// TIA Portal project "PID_Tank_V17" (V17)

(* hardware
DEVICE "S7-1200 station_1"  S7-1200 Station
   slot 0: "Rack_0"  S7-1200 Rack  Rack  V1.0
   slot 1: "PLC_1"  CPU 1215C DC/DC/DC  6ES7 215-1AG40-0XB0  V4.4
DEVICE "HMI_1"  KTP700 Basic PN
   slot 0: "HMI_1"  KTP700 Basic PN  6AV2 123-2GB03-0AX0  16.0.0.0
   slot 1: "HMI_RT_1"  KTP700 Basic PN  6AV2 123-2GB03-0AX0  16.0.0.0
   slot 5: "HMI_1.IE_CP_1"  PROFINET Interface  16.0.0.0
      slot 1: "PROFINET Interface_1"  PROFINET Interface
         slot 1: "Port_1"  Port
*)

// ===== PLC "PLC_1"  CPU 1215C DC/DC/DC =====

VAR_GLOBAL   // PLC tag table "Default tag table"
   "IW_TankLevel_Sensor" AT %ID30 : Real;
   "IW_Flow_Sensor" AT %ID34 : Real;
   "Q_Hooter" AT %Q0.0 : Bool;
   "QW_DrainValve_Signal" AT %QD34 : Real;
   "QW_FillingValve_Signal" AT %QD30 : Real;
END_VAR

DATA_BLOCK "FB_PID_DB"   // DB5
{ S7_Optimized_Access := 'TRUE' }
VERSION : 0.1
// stored: InstanceOfName FB_PID
"FB_PID"
BEGIN
END_DATA_BLOCK

// folder: Global DB

DATA_BLOCK "DB_System"   // DB2
{ S7_Optimized_Access := 'TRUE' }
VERSION : 0.1
   VAR
      "ActualValue_%" : Real;
      "ProcessVAlue_PV_%" : Real;
   END_VAR
BEGIN
END_DATA_BLOCK

DATA_BLOCK "DB_Alarm"   // DB3
{ S7_Optimized_Access := 'TRUE' }
VERSION : 0.1
BEGIN
END_DATA_BLOCK

DATA_BLOCK "DB_HMI_Interface"   // DB4
{ S7_Optimized_Access := 'TRUE' }
VERSION : 0.1
   VAR
      From_HMI_To_PLC : Struct
         "SetValue_SP_%" : Real;
         ki : Real;
         kp : Real;
         kd : Real;
         Auto : Bool;
         DrainValve_SetPoint : Real;
         AlarmBit : Bool;
      END_STRUCT;
      From_PLC_To_HMI : Struct
         ActualValue : Real;
         SetValue_SP_InRange : Real;
         "ActualValue_%" : Real;
         "Error_%" : Real;
         Error_InRange : Real;
         Filling_Pipe_Animation_SetPoint : Int;
         P_Term : Real;
         I_Term : Real;
         D_Term : Real;
         FillingValve_SetPoint : Real;
      END_STRUCT;
      Alarm : Word;
   END_VAR
BEGIN
END_DATA_BLOCK

// folder: IO_mapping

DATA_BLOCK "DB_IO_Mapping"   // DB1
{ S7_Optimized_Access := 'TRUE' }
VERSION : 0.1
   VAR
      Input : Struct
         IW_TankLevel_Sensor : Real;
         IW_Flow_Sensor : Real;
      END_STRUCT;
      Output : Struct
         Q_Hooter : Bool;
         QW_DrainValve_Signal : Real;
         QW_FillingValve_Signal : Real;
      END_STRUCT;
   END_VAR
BEGIN
END_DATA_BLOCK

// folder: (top level)

ORGANIZATION_BLOCK "Main"   // OB1, LAD, ProgramCycle
TITLE = "Main Program Sweep (Cycle)"
{ S7_Optimized_Access := 'TRUE' }
VERSION : 0.1
   VAR_INPUT
      Initial_Call : Bool;   // Initial call of this OB
      Remanence : Bool;   // =True, if remanent data are available
   END_VAR
BEGIN

REGION Network 1: Factory IO Connection
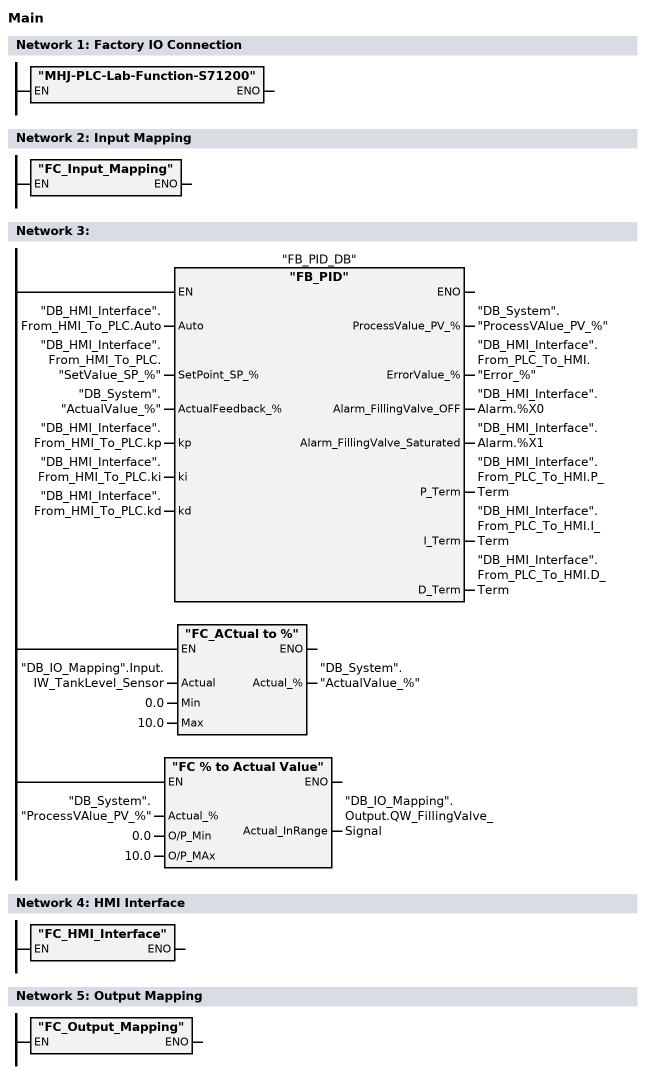
   RUNG wire#powerrail
      "MHJ-PLC-Lab-Function-S71200"()
   END_RUNG
   // the same network as SCL:
   "MHJ-PLC-Lab-Function-S71200"();
END_REGION

REGION Network 2: Input Mapping
   RUNG wire#powerrail
      "FC_Input_Mapping"()
   END_RUNG
   // the same network as SCL:
   "FC_Input_Mapping"();
END_REGION

REGION Network 3
   RUNG wire#powerrail
      "FB_PID_DB"(Auto := "DB_HMI_Interface".From_HMI_To_PLC.Auto, "SetPoint_SP_%" := "DB_HMI_Interface".From_HMI_To_PLC."SetValue_SP_%", "ActualFeedback_%" := "DB_System"."ActualValue_%", kp := "DB_HMI_Interface".From_HMI_To_PLC.kp, ki := "DB_HMI_Interface".From_HMI_To_PLC.ki, kd := "DB_HMI_Interface".From_HMI_To_PLC.kd, "ProcessValue_PV_%" => "DB_System"."ProcessVAlue_PV_%", "ErrorValue_%" => "DB_HMI_Interface".From_PLC_To_HMI."Error_%", Alarm_FillingValve_OFF => "DB_HMI_Interface".Alarm.%X0, Alarm_FillingValve_Saturated => "DB_HMI_Interface".Alarm.%X1, P_Term => "DB_HMI_Interface".From_PLC_To_HMI.P_Term, I_Term => "DB_HMI_Interface".From_PLC_To_HMI.I_Term, D_Term => "DB_HMI_Interface".From_PLC_To_HMI.D_Term)
   END_RUNG
   RUNG wire#powerrail
      "FC_ACtual to %"(Actual := "DB_IO_Mapping".Input.IW_TankLevel_Sensor, Min := 0.0, Max := 10.0, "Actual_%" => "DB_System"."ActualValue_%")
   END_RUNG
   RUNG wire#powerrail
      "FC % to Actual Value"("Actual_%" := "DB_System"."ProcessVAlue_PV_%", "O/P_Min" := 0.0, "O/P_MAx" := 10.0, Actual_InRange => "DB_IO_Mapping".Output.QW_FillingValve_Signal)
   END_RUNG
   // the same network as SCL:
   "FB_PID_DB"(Auto := "DB_HMI_Interface".From_HMI_To_PLC.Auto,   // "FB_PID"
               "SetPoint_SP_%" := "DB_HMI_Interface".From_HMI_To_PLC."SetValue_SP_%",
               "ActualFeedback_%" := "DB_System"."ActualValue_%",
               kp := "DB_HMI_Interface".From_HMI_To_PLC.kp,
               ki := "DB_HMI_Interface".From_HMI_To_PLC.ki,
               kd := "DB_HMI_Interface".From_HMI_To_PLC.kd,
               "ProcessValue_PV_%" => "DB_System"."ProcessVAlue_PV_%",
               "ErrorValue_%" => "DB_HMI_Interface".From_PLC_To_HMI."Error_%",
               Alarm_FillingValve_OFF => "DB_HMI_Interface".Alarm.%X0,
               Alarm_FillingValve_Saturated => "DB_HMI_Interface".Alarm.%X1,
               P_Term => "DB_HMI_Interface".From_PLC_To_HMI.P_Term,
               I_Term => "DB_HMI_Interface".From_PLC_To_HMI.I_Term,
               D_Term => "DB_HMI_Interface".From_PLC_To_HMI.D_Term);
   "FC_ACtual to %"(Actual := "DB_IO_Mapping".Input.IW_TankLevel_Sensor,
                    Min := 0.0,
                    Max := 10.0,
                    "Actual_%" => "DB_System"."ActualValue_%");
   "FC % to Actual Value"("Actual_%" := "DB_System"."ProcessVAlue_PV_%",
                          "O/P_Min" := 0.0,
                          "O/P_MAx" := 10.0,
                          Actual_InRange => "DB_IO_Mapping".Output.QW_FillingValve_Signal);
END_REGION

REGION Network 4: HMI Interface
   RUNG wire#powerrail
      "FC_HMI_Interface"()
   END_RUNG
   // the same network as SCL:
   "FC_HMI_Interface"();
END_REGION

REGION Network 5: Output Mapping
   RUNG wire#powerrail
      "FC_Output_Mapping"()
   END_RUNG
   // the same network as SCL:
   "FC_Output_Mapping"();
END_REGION
END_ORGANIZATION_BLOCK

// folder: FB_Library

FUNCTION_BLOCK "FB_PID"   // FB1, SCL
{ S7_Optimized_Access := 'TRUE' }
VERSION : 0.1
   VAR_INPUT
      Auto : Bool;
      "SetPoint_SP_%" : Real;
      "ActualFeedback_%" : Real;
      kp : Real;
      ki : Real;
      kd : Real;
   END_VAR
   VAR_OUTPUT
      "ProcessValue_PV_%" : Real;
      "ErrorValue_%" : Real;
      Alarm_FillingValve_OFF : Bool;
      Alarm_FillingValve_Saturated : Bool;
      P_Term : Real;
      I_Term : Real;
      D_Term : Real;
   END_VAR
   VAR
      Prev_Error : Real;
      IntegralError : Real;
      IntegralReset : Bool;
      FiilingValve_OFF_TONStart_Condition : Bool;
      FillingValve_Saturated_TONStart_Condition : Bool;
      IEC_Timer_0_Instance_FillingValve_OFF : TON_TIME;
      IEC_Timer_0_Instance_FillingValve_Saturated : TON_TIME;
   END_VAR
   VAR_TEMP
      p_Term_Temp : Real;
      i_Term_Temp : Real;
      d_Term_Temp : Real;
      Current_Error_Temp : Real;
      processed_Value_Temp : Real;
   END_VAR
BEGIN


   IF #Auto THEN

       #Current_Error_Temp :=  #"SetPoint_SP_%" - #"ActualFeedback_%" ;

       //P-Term Calculation
       #p_Term_Temp:= #Current_Error_Temp * #kp;

       //I-Term Calculation
       #i_Term_Temp := (#IntegralError + #Current_Error_Temp) * #ki;

       //D-Term Calculation
       #d_Term_Temp := ( #Current_Error_Temp - #Prev_Error) * #kd;

       //Process Value
       #processed_Value_Temp  := #p_Term_Temp + #i_Term_Temp + #d_Term_Temp;

       //Make Range 0-100
       IF #processed_Value_Temp > 100 THEN
           #processed_Value_Temp := 100;
       ELSIF #processed_Value_Temp < 0 THEN
           #processed_Value_Temp := 0;
       END_IF;


       //Alarm Detection

       //Filling Valve OFF
       IF (#"ActualFeedback_%" < #"SetPoint_SP_%") & (#Current_Error_Temp >= #Prev_Error) THEN
           #FiilingValve_OFF_TONStart_Condition := TRUE;
       ELSE
           #FiilingValve_OFF_TONStart_Condition := FALSE;
       END_IF;

       //Make timer On or OFF
       IF #FiilingValve_OFF_TONStart_Condition THEN
           #IEC_Timer_0_Instance_FillingValve_OFF(IN:=TRUE,
                         PT:=T#30s);
       ELSE
           #IEC_Timer_0_Instance_FillingValve_OFF(IN := FALSE,
                                 PT := T#30s);
       END_IF;
       //IF timer On than Set Alarm
       IF #IEC_Timer_0_Instance_FillingValve_OFF.Q THEN
           #Alarm_FillingValve_OFF := TRUE;
       ELSE
           #Alarm_FillingValve_OFF := FALSE;
       END_IF;

       //Filling Valve Saturated Alarm
       IF (#"ActualFeedback_%" > #"SetPoint_SP_%") & (#Current_Error_Temp <= #Prev_Error) THEN
           #FillingValve_Saturated_TONStart_Condition := TRUE;
       ELSE
           #FillingValve_Saturated_TONStart_Condition := FALSE;
       END_IF;

       IF #FillingValve_Saturated_TONStart_Condition THEN
           #IEC_Timer_0_Instance_FillingValve_Saturated(IN := TRUE,
                                                        PT := T#30s);
       ELSE
           #IEC_Timer_0_Instance_FillingValve_Saturated(IN := FALSE,
                                                        PT := T#30s);
       END_IF;

       IF #IEC_Timer_0_Instance_FillingValve_Saturated.Q THEN
           #Alarm_FillingValve_Saturated := TRUE;
       ELSE
           #Alarm_FillingValve_Saturated := FALSE;
       END_IF;



       //------------------------
       //Write to O/P
       #"ProcessValue_PV_%" := #processed_Value_Temp;
       #"ErrorValue_%" := #Current_Error_Temp;
       #P_Term := #p_Term_Temp;
       #I_Term := #i_Term_Temp;
       #D_Term := #d_Term_Temp;

       //Write State data
       #Prev_Error := #Current_Error_Temp;
       #IntegralError := #IntegralError + #Current_Error_Temp;


   ELSE
       #IntegralError := 0;
       #Prev_Error := 0;
       #IntegralReset := 0;
       #FiilingValve_OFF_TONStart_Condition := FALSE;
       #FillingValve_Saturated_TONStart_Condition := FALSE;
       #"ProcessValue_PV_%" := 0;
       #P_Term := 0;
       #I_Term := 0;
       #D_Term := 0;
       #Alarm_FillingValve_OFF := FALSE;
       #Alarm_FillingValve_Saturated := FALSE;
   END_IF;
END_FUNCTION_BLOCK

// folder: FC_Library

FUNCTION "FC_HMI_Interface" : Void   // FC3, SCL
{ S7_Optimized_Access := 'TRUE' }
VERSION : 0.1
   VAR_TEMP
      Norm_Data : Real;
   END_VAR
BEGIN

   #Norm_Data := NORM_X(MIN := 0.0, VALUE := "DB_IO_Mapping".Input.IW_TankLevel_Sensor, MAX := 10.0);

   "DB_HMI_Interface".From_PLC_To_HMI.ActualValue := SCALE_X(MIN := 0.0, VALUE := #Norm_Data, MAX := 300.0);
   "DB_HMI_Interface".From_PLC_To_HMI.Filling_Pipe_Animation_SetPoint := REAL_TO_INT("DB_HMI_Interface".From_PLC_To_HMI.ActualValue);
   "DB_HMI_Interface".From_PLC_To_HMI."ActualValue_%" := SCALE_X(MIN := 0.0, VALUE := #Norm_Data, MAX := 100.0);

   IF "DB_HMI_Interface".From_HMI_To_PLC.Auto THEN
       "DB_IO_Mapping".Output.QW_DrainValve_Signal := "DB_HMI_Interface".From_HMI_To_PLC.DrainValve_SetPoint;
   ELSE
       "DB_IO_Mapping".Output.QW_DrainValve_Signal := 0.0;
   END_IF;
   "DB_HMI_Interface".From_PLC_To_HMI.SetValue_SP_InRange := SCALE_X(MIN := 0.0, VALUE := "DB_HMI_Interface".From_HMI_To_PLC."SetValue_SP_%", MAX := 3.0);
   "DB_HMI_Interface".From_PLC_To_HMI."ActualValue_%" := "DB_System"."ActualValue_%";
   "DB_HMI_Interface".From_PLC_To_HMI.Error_InRange := SCALE_X(MIN := 0.0, VALUE := "DB_HMI_Interface".From_PLC_To_HMI."Error_%" , MAX := 3.0);

   "DB_HMI_Interface".From_PLC_To_HMI.FillingValve_SetPoint := "DB_IO_Mapping".Output.QW_FillingValve_Signal;

   "DB_IO_Mapping".Output.Q_Hooter := "DB_HMI_Interface".From_HMI_To_PLC.AlarmBit;
END_FUNCTION

FUNCTION "FC_ACtual to %" : Void   // FC4, SCL
{ S7_Optimized_Access := 'TRUE' }
VERSION : 0.1
   VAR_INPUT
      Actual : Real;
      Min : Real;
      Max : Real;
   END_VAR
   VAR_OUTPUT
      "Actual_%" : Real;
   END_VAR
   VAR_TEMP
      Norm_Value : Real;
   END_VAR
BEGIN
   #Norm_Value:=NORM_X(MIN:=#Min, VALUE:=#Actual, MAX:=#Max);
   #"Actual_%" := SCALE_X(MIN := 0.0, VALUE := #Norm_Value, MAX := 100.0);
END_FUNCTION

FUNCTION "FC % to Actual Value" : Void   // FC5, SCL
{ S7_Optimized_Access := 'TRUE' }
VERSION : 0.1
   VAR_INPUT
      "Actual_%" : Real;
      "O/P_Min" : Real;
      "O/P_MAx" : Real;
   END_VAR
   VAR_OUTPUT
      Actual_InRange : Real;
   END_VAR
   VAR_TEMP
      Norm_Value : Real;
   END_VAR
BEGIN
   #Norm_Value := NORM_X(MIN := 0.0, VALUE := #"Actual_%", MAX := 100.0);
   #Actual_InRange := SCALE_X(MIN := #"O/P_Min", VALUE := #Norm_Value, MAX := #"O/P_MAx");
END_FUNCTION

FUNCTION "MHJ-PLC-Lab-Function-S71200" : Void   // FC9000, SCL
{ S7_Optimized_Access := 'TRUE' }
VERSION : 0.1
   VAR_TEMP
      rdTimeReturn : Int;
      outputTime : DTL;
      SyncVal : Byte;
      forVal : Int;
      forVal_2 : Int;
      Value : Byte;
   END_VAR
   VAR CONSTANT
      CompVal : Byte := 16#34;
      Value_01 : Byte := 16#11;
      Value_01_DW : DWord := 16#A165_D992;
      Value_02_DW : DWord := 16#58BE_4401;
   END_VAR
BEGIN

   #Value:=PEEK(area := 16#82,
        dbNumber := 0,
        byteOffset := 511);
   #Value := #Value + 1;

   POKE(area := 16#82,
        dbNumber := 0,
        byteOffset := 511,
        value := #Value);

   POKE(area:=16#81,
        dbNumber:=0,
        byteOffset:=1016,
        value:=#Value_01_DW);
   POKE(area := 16#81,
        dbNumber := 0,
        byteOffset := 1020,
        value := #Value_02_DW);

   POKE(area := 16#81,
        dbNumber := 0,
        byteOffset := 511,
        value := B#16#00);

   FOR #forVal := 0 TO 500 DO
       FOR #forVal_2:=0 TO 10 DO
           #rdTimeReturn:=RD_SYS_T(#outputTime);
           #rdTimeReturn := WR_SYS_T(#outputTime);
           #rdTimeReturn := RD_SYS_T(#outputTime);
           #rdTimeReturn := WR_SYS_T(#outputTime);
       END_FOR;
       #SyncVal:= PEEK(area := 16#81,
                      dbNumber := 0,
                      byteOffset := 511);
       IF #SyncVal = #CompVal THEN
          GOTO M_1;
       END_IF;
   END_FOR;
   RETURN;

   M_1:
   POKE(area := 16#81,
        dbNumber := 0,
        byteOffset := 511,
        value := B#16#0);
END_FUNCTION

// folder: IO_mapping

FUNCTION "FC_Input_Mapping" : Void   // FC1, SCL
{ S7_Optimized_Access := 'TRUE' }
VERSION : 0.1
   VAR_TEMP
      ScaledData : Real;
   END_VAR
BEGIN

   "DB_IO_Mapping".Input.IW_TankLevel_Sensor := "IW_TankLevel_Sensor";
   "DB_IO_Mapping".Input.IW_Flow_Sensor := "IW_Flow_Sensor";
END_FUNCTION

FUNCTION "FC_Output_Mapping" : Void   // FC2, SCL
{ S7_Optimized_Access := 'TRUE' }
VERSION : 0.1
BEGIN

   "Q_Hooter" := "DB_IO_Mapping".Output.Q_Hooter;
   "QW_DrainValve_Signal" := "DB_IO_Mapping".Output.QW_DrainValve_Signal;
   "QW_FillingValve_Signal" := "DB_IO_Mapping".Output.QW_FillingValve_Signal;
END_FUNCTION

(* ===== HMI "HMI_RT_1" =====
system functions are stored by id; their names below are inferred from use
connection "HMI_Connection_1": ETHERNET, SMART_S7_1200_OMS

HMI tags "Default tag table"
   "Tag_ScreenNumber" : UInt, internal
   "DB_HMI_Interface_From_HMI_To_PLC_SetValue_SP_%" : Real = PLC DB_HMI_Interface.From_HMI_To_PLC.SetValue_SP_%, 1 s
   "DB_HMI_Interface_From_PLC_To_HMI_ActualValue_%" : Real = PLC DB_HMI_Interface.From_PLC_To_HMI.ActualValue_%, 1 s
   "DB_HMI_Interface_From_PLC_To_HMI_ActualValue_PV" : Real = PLC DB_HMI_Interface.From_PLC_To_HMI.ActualValue, 1 s
   "DB_HMI_Interface_From_PLC_To_HMI_Error_%" : Real = PLC DB_HMI_Interface.From_PLC_To_HMI.Error_%, 1 s
   "DB_HMI_Interface_From_PLC_To_HMI_Error_InRange" : Real = PLC DB_HMI_Interface.From_PLC_To_HMI.Error_InRange, 1 s
   "DB_HMI_Interface_From_HMI_To_PLC_ki" : Real = PLC DB_HMI_Interface.From_HMI_To_PLC.ki, 1 s
   "DB_HMI_Interface_From_HMI_To_PLC_kp" : Real = PLC DB_HMI_Interface.From_HMI_To_PLC.kp, 1 s
   "DB_HMI_Interface_From_HMI_To_PLC_kd" : Real = PLC DB_HMI_Interface.From_HMI_To_PLC.kd, 1 s
   "DB_HMI_Interface_From_HMI_To_PLC_DrainValve_SetPoint" : Real = PLC DB_HMI_Interface.From_HMI_To_PLC.DrainValve_SetPoint, 1 s
   "DB_HMI_Interface_From_HMI_To_PLC_Auto" : Bool = PLC DB_HMI_Interface.From_HMI_To_PLC.Auto, 1 s
   "DB_HMI_Interface_From_PLC_To_HMI_SetValue_SP_InRange" : Real = PLC DB_HMI_Interface.From_PLC_To_HMI.SetValue_SP_InRange, 100 ms
   "DB_HMI_Interface_From_PLC_To_HMI_Filling_Valve_SetPoint" : Int = PLC DB_HMI_Interface.From_PLC_To_HMI.Filling_Pipe_Animation_SetPoint, 1 s
   "DB_HMI_Interface_From_PLC_To_HMI_FillingValve_SetPoint" : Real = PLC DB_HMI_Interface.From_PLC_To_HMI.FillingValve_SetPoint, 1 s
   "DB_HMI_Interface_From_PLC_To_HMI_P_Term" : Real = PLC DB_HMI_Interface.From_PLC_To_HMI.P_Term, 1 s
   "DB_HMI_Interface_From_PLC_To_HMI_I_Term" : Real = PLC DB_HMI_Interface.From_PLC_To_HMI.I_Term, 1 s
   "DB_HMI_Interface_From_PLC_To_HMI_D_Term" : Real = PLC DB_HMI_Interface.From_PLC_To_HMI.D_Term, 1 s
   "DB_HMI_Interface_Alarm" : Word = PLC DB_HMI_Interface.Alarm, 1 s
   "DB_HMI_Interface_From_HMI_To_PLC_AlarmBit" : Bool = PLC DB_HMI_Interface.From_HMI_To_PLC.AlarmBit, 1 s

discrete alarms
   1: 'Filling Valve Failure Detected- Valave OFF', class Errors, trigger "DB_HMI_Interface_Alarm" bit 0
      on Coming: SetBit("DB_HMI_Interface_From_HMI_To_PLC_AlarmBit")
      on Going: ResetBit("DB_HMI_Interface_From_HMI_To_PLC_AlarmBit")
      on Acknowledge: ResetBit("DB_HMI_Interface_From_HMI_To_PLC_AlarmBit")
   2: 'Filling Valve Failure Detected- Valave Saturated', class Errors, trigger "DB_HMI_Interface_Alarm" bit 1
      on Coming: SetBit("DB_HMI_Interface_From_HMI_To_PLC_AlarmBit")
      on Going: ResetBit("DB_HMI_Interface_From_HMI_To_PLC_AlarmBit")
      on Acknowledge: ResetBit("DB_HMI_Interface_From_HMI_To_PLC_AlarmBit")

analog alarms
   1: 'Level High Detected', class Warnings, trigger "DB_HMI_Interface_From_PLC_To_HMI_ActualValue_%"
   2: 'Level Critical High Detected', class Errors, trigger "DB_HMI_Interface_From_PLC_To_HMI_ActualValue_%"
      on Coming: SetBit("DB_HMI_Interface_From_HMI_To_PLC_AlarmBit")
      on Going: ResetBit("DB_HMI_Interface_From_HMI_To_PLC_AlarmBit")
      on Acknowledge: ResetBit("DB_HMI_Interface_From_HMI_To_PLC_AlarmBit")
   3: 'Level Low Detected', class Warnings, trigger "DB_HMI_Interface_From_PLC_To_HMI_ActualValue_%"
   4: 'Level Critical Low Detected', class Errors, trigger "DB_HMI_Interface_From_PLC_To_HMI_ActualValue_%"
      on Coming: SetBit("DB_HMI_Interface_From_HMI_To_PLC_AlarmBit")
      on Going: ResetBit("DB_HMI_Interface_From_HMI_To_PLC_AlarmBit")
      on Acknowledge: ResetBit("DB_HMI_Interface_From_HMI_To_PLC_AlarmBit")

Template "Template_1" 800x480
   DateTimeField "HmiScreenItemData" at 695,25 size 105x25
   DateTimeField "HmiScreenItemData_1" at 695,0 size 105x25
   GraphicView "Logo" at 0,0 size 91x51; Picture "Logo of HMI_1"

screen "Root screen" 800x480, template "Template_1"
   on GenerateScreen: SetTag("Tag_ScreenNumber", 1)
   Bar "Bar_1" at 529,285 size 141x185; MinimumValue 0; MaximumValue 300
      ProcessValue <- "DB_HMI_Interface_From_PLC_To_HMI_ActualValue_PV"
   Rectangle "Rectangle_5" at 609,211 size 17x257
      Appearance <- "DB_HMI_Interface_From_PLC_To_HMI_FillingValve_SetPoint"
   Rectangle "Rectangle_1" at 348,451 size 96x14
      Appearance <- "DB_HMI_Interface_From_HMI_To_PLC_DrainValve_SetPoint"
   GraphicView "Graphic view_2" at 654,137 size 45x61; Picture "Graphic_2"
   GraphicView "Graphic view_3" at 443,411 size 45x61; Picture "Graphic_2"
   Rectangle "Rectangle_3" at 485,450 size 43x14
      Appearance <- "DB_HMI_Interface_From_PLC_To_HMI_ActualValue_PV"
   IOField "I/O field_1" at 112,132 size 96x32; FormatPattern 999.99
      ProcessValue <- "DB_HMI_Interface_From_HMI_To_PLC_SetValue_SP_%"
   IOField "I/O field_2" at 112,174 size 96x32; FormatPattern 999.99
      ProcessValue <- "DB_HMI_Interface_From_PLC_To_HMI_ActualValue_%"
   IOField "I/O field_3" at 112,216 size 96x32; FormatPattern 999.99
      ProcessValue <- "DB_HMI_Interface_From_PLC_To_HMI_Error_%"
   IOField "I/O field_4" at 428,373 size 65x32; FormatPattern 999.99
      ProcessValue <- "DB_HMI_Interface_From_HMI_To_PLC_DrainValve_SetPoint"
   IOField "I/O field_5" at 651,103 size 65x32; FormatPattern 999.99
      ProcessValue <- "DB_HMI_Interface_From_PLC_To_HMI_FillingValve_SetPoint"
   IOField "I/O field_6" at 698,358 size 70x32; FormatPattern 999.9
      ProcessValue <- "DB_HMI_Interface_From_PLC_To_HMI_ActualValue_PV"
   IOField "I/O field_7" at 112,304 size 96x32; FormatPattern 999.99
      ProcessValue <- "DB_HMI_Interface_From_HMI_To_PLC_kp"
   IOField "I/O field_8" at 112,346 size 96x32; FormatPattern 999.99
      ProcessValue <- "DB_HMI_Interface_From_HMI_To_PLC_ki"
   TextField "Text field_4" at 75,305 size 30x25; Text 'p'
   TextField "Text field_5" at 74,348 size 30x25; Text 'i'
   TextField "Text field_1" at 26,134 size 79x25; Text 'SetValue'
   TextField "Text field_2" at 44,179 size 61x25; Text 'Actual'
   TextField "Text field_3" at 47,216 size 58x25; Text 'Error'
   TextField "Text field_6" at 76,392 size 30x25; Text 'd'
   IOField "I/O field_9" at 112,389 size 96x32; FormatPattern 999.99
      ProcessValue <- "DB_HMI_Interface_From_HMI_To_PLC_kd"
   IOField "I/O field_10" at 218,174 size 96x32; FormatPattern 999.9
      ProcessValue <- "DB_HMI_Interface_From_PLC_To_HMI_ActualValue_PV"
   IOField "I/O field_11" at 219,133 size 96x32; FormatPattern 999.9
      ProcessValue <- "DB_HMI_Interface_From_PLC_To_HMI_SetValue_SP_InRange"
   IOField "I/O field_12" at 219,215 size 96x32; FormatPattern 999.99
      ProcessValue <- "DB_HMI_Interface_From_PLC_To_HMI_Error_InRange"
   Switch "Switch_1" at 357,107 size 162x32; CaptionText 'Switch'; TextOff 'Manual'; TextOn 'Auto'
      ProcessValue <- "DB_HMI_Interface_From_HMI_To_PLC_Auto"
   TextField "Text field_7" at 118,102 size 78x25; Text 'Value %'
   TextField "Text field_8" at 213,102 size 110x25; Text 'Value Range'
   Rectangle "Rectangle_6" at 590,286 size 10x183
      VerticalMovement <- "DB_HMI_Interface_From_PLC_To_HMI_Filling_Valve_SetPoint"
      Appearance <- "DB_HMI_Interface_From_PLC_To_HMI_FillingValve_SetPoint"
   GraphicView "Graphic view_1" at 515,246 size 169x44; Picture "Graphic_1"
   Rectangle "Rectangle_4" at 619,175 size 36x15
      Appearance <- "DB_HMI_Interface_From_PLC_To_HMI_FillingValve_SetPoint"
   Rectangle "Rectangle_7" at 588,210 size 16x38
      Appearance <- "DB_HMI_Interface_From_PLC_To_HMI_FillingValve_SetPoint"
   GraphicView "Graphic view_4" at 569,159 size 54x52; Picture "Graphic_3"
   IOField "I/O field_13" at 217,304 size 96x32; FormatPattern 999.9
      ProcessValue <- "DB_HMI_Interface_From_PLC_To_HMI_P_Term"
   IOField "I/O field_14" at 217,346 size 96x32; FormatPattern 999.9
      ProcessValue <- "DB_HMI_Interface_From_PLC_To_HMI_I_Term"
   IOField "I/O field_15" at 218,389 size 96x32; FormatPattern 999.9
      ProcessValue <- "DB_HMI_Interface_From_PLC_To_HMI_D_Term"
   TextField "Text field_9" at 101,275 size 78x25; Text 'gain'
   TextField "Text field_10" at 200,276 size 125x25; Text 'derived value'
   Button "Button_1" at 699,53 size 96x32; TextOff 'Alarm'; PictureOff "Right_Arrow"
      on Click: ActivateScreen("Screen_1", 0)
   TextField "Text field_11" at 655,282 size 42x25; Text '300'
   TextField "Text field_12" at 655,364 size 42x25; Text '150'
   TextField "Text field_13" at 642,451 size 42x25; Text '0'

screen "Screen_1" 800x480
   AlarmView "Alarm view_1" at 14,40 size 768x346
   Button "Button_1" at 14,403 size 96x72; TextOff 'Home'; PictureOff "Home"
      on Click: ActivateScreen("Root screen", 0)
*)